(*~
<docu>
	<summary>
			Allows to concat strings using fluent interface. It's similar to C# StringBuilder class
			Usage as follows :
			<code>
				ErrorString := _stringBuilder
					.Clear()
					.Append('Error number: ')
					.Append(INT_TO_STRING(ErrorNumber))
					.Append('. Message: ')
					.Append(ErrorMessage)
					.Append('.')
					.ToString();
			</code>
			
			Inspired by Gerhard Barteling blogpost at https://www.plccoder.com/fluent-code/
	</summary>				
</docu>	
~*)	
FUNCTION_BLOCK StringBuilder
VAR
	{attribute 'hide'}
    _workString:STRING(255);
END_VAR

(*
	Thanks to https://github.com/bengeisler/TcLog
*)

METHOD PROTECTED AnyToString : STRING(255)
VAR_INPUT
	Data:	ANY;
END_VAR
VAR
	pAnyBOOL		: POINTER TO BOOL; 
	pAnyBYTE		: POINTER TO BYTE; 
	pAnyWORD		: POINTER TO WORD; 
	pAnyDWORD		: POINTER TO DWORD;
	pAnyLWORD		: POINTER TO LWORD;
	pAnySINT		: POINTER TO SINT; 
	pAnyUSINT		: POINTER TO USINT;
	pAnyINT			: POINTER TO INT;  
	pAnyUINT		: POINTER TO UINT; 
	pAnyDINT		: POINTER TO DINT; 
	pAnyUDINT		: POINTER TO UDINT;
	pAnyLINT		: POINTER TO LINT; 
	pAnyULINT		: POINTER TO ULINT;
	pAnyLTIME		: POINTER TO LTIME;	
	pAnyReal 		: POINTER TO REAL;
	pAnyLReal		: POINTER TO LREAL;	
	pAnyDateAndTime : POINTER TO DATE_AND_TIME;
	pAnyDate		: POINTER TO DATE;
	pAnyTime		: POINTER TO TIME;
	pAnyWString		: POINTER TO WSTRING;
	pAnyTOD			: POINTER TO TOD;
	pAnyString		: POINTER TO STRING;	
	sString			: T_MAXSTRING;
	wWString		: WSTRING;
END_VAR
IF Data.TypeClass = __SYSTEM.TYPE_CLASS.TYPE_REAL THEN
	pAnyReal := Data.pValue;
	AnyToString := REAL_TO_STRING(pAnyReal^);
	
ELSIF Data.TypeClass = __SYSTEM.TYPE_CLASS.TYPE_LREAL THEN
	pAnyLReal := Data.pValue;
	AnyToString := LREAL_TO_STRING(pAnyLReal^);
	
ELSIF Data.TypeClass = __SYSTEM.TYPE_CLASS.TYPE_DATEANDTIME THEN
	pAnyDateAndTime := Data.pValue;
	AnyToString := DT_TO_STRING(pAnyDateAndTime^);	
	
ELSIF Data.TypeClass = __SYSTEM.TYPE_CLASS.TYPE_DATE THEN
	pAnyDate := Data.pValue;
	AnyToString := DATE_TO_STRING(pAnyDate^);
	
ELSIF Data.TypeClass = __SYSTEM.TYPE_CLASS.TYPE_TIME THEN
	pAnyTime := Data.pValue;
	AnyToString := TIME_TO_STRING(pAnyTime^);
	
ELSIF Data.TypeClass = __SYSTEM.TYPE_CLASS.TYPE_STRING THEN
	pAnyString := Data.pValue;
	AnyToString := pAnyString^;
	
ELSIF Data.TypeClass = __SYSTEM.TYPE_CLASS.TYPE_WSTRING THEN
	pAnyWString := Data.pValue;
	wWString := pAnyWString^;
	WSTRING_TO_STRING2(ADR(sString), ADR(wWstring), SIZEOF(wWString));
	AnyToString := sString;
	
ELSIF Data.TypeClass = __SYSTEM.TYPE_CLASS.TYPE_TIMEOFDAY THEN
	pAnyTOD := Data.pValue;
	AnyToString := TOD_TO_STRING(pAnyTOD^);
ELSIF Data.TypeClass = __SYSTEM.TYPE_CLASS.TYPE_BOOL THEN 	
	pAnyBOOL := Data.pValue;
	AnyToString := BOOL_TO_STRING(pAnyBool^);
ELSIF Data.TypeClass = __SYSTEM.TYPE_CLASS.TYPE_BYTE THEN
	pAnyBYTE := Data.pValue;
	AnyToString := BYTE_TO_STRING(pAnyBYTE^);	
ELSIF Data.TypeClass = __SYSTEM.TYPE_CLASS.TYPE_WORD THEN
	pAnyWORD := Data.pValue;
	AnyToString := WORD_TO_STRING(pAnyWORD^);	
ELSIF Data.TypeClass = __SYSTEM.TYPE_CLASS.TYPE_DWORD THEN
	pAnyDWORD := Data.pValue;	
	AnyToString := DWORD_TO_STRING(pAnyDWORD^);
ELSIF Data.TypeClass = __SYSTEM.TYPE_CLASS.TYPE_LWORD THEN
	pAnyLWORD := Data.pValue;	
	AnyToString := LWORD_TO_STRING(pAnyLWORD^);
ELSIF Data.TypeClass = __SYSTEM.TYPE_CLASS.TYPE_SINT THEN
	pAnySINT := Data.pValue;	
	AnyToString := SINT_TO_STRING(pAnySINT^);					
ELSIF Data.TypeClass = __SYSTEM.TYPE_CLASS.TYPE_USINT THEN
	pAnyUSINT := Data.pValue;	
	AnyToString := USINT_TO_STRING(pAnyUSINT^);	
ELSIF Data.TypeClass = __SYSTEM.TYPE_CLASS.TYPE_INT THEN
	pAnyINT := Data.pValue;	
	AnyToString := INT_TO_STRING(pAnyINT^);	
ELSIF Data.TypeClass = __SYSTEM.TYPE_CLASS.TYPE_UINT THEN
	pAnyUINT := Data.pValue;	
	AnyToString := UINT_TO_STRING(pAnyUINT^);	
ELSIF Data.TypeClass = __SYSTEM.TYPE_CLASS.TYPE_DINT THEN
	pAnyDINT := Data.pValue;	
	AnyToString := DINT_TO_STRING(pAnyDINT^);	
ELSIF Data.TypeClass = __SYSTEM.TYPE_CLASS.TYPE_UDINT THEN
	pAnyUDINT := Data.pValue;	
	AnyToString := UDINT_TO_STRING(pAnyUDINT^);	
ELSIF Data.TypeClass = __SYSTEM.TYPE_CLASS.TYPE_LINT THEN
	pAnyLINT := Data.pValue;	
	AnyToString := LINT_TO_STRING(pAnyLINT^);	
ELSIF Data.TypeClass = __SYSTEM.TYPE_CLASS.TYPE_ULINT THEN
	pAnyULINT := Data.pValue;	
	AnyToString := ULINT_TO_STRING(pAnyULINT^);	
ELSIF Data.TypeClass = __SYSTEM.TYPE_CLASS.TYPE_LTIME THEN
	pAnyLTIME := Data.pValue;	
	AnyToString := LTIME_TO_STRING(pAnyLTIME^);		
ELSE	
	AnyToString := ANY_TO_STRING(Data.pValue^);
END_IF
END_METHOD

METHOD Append : REFERENCE TO StringBuilder
VAR_INPUT
    Text :STRING(255); 
END_VAR
_workString := Concat(_workString,text);
Append REF= THIS^;
END_METHOD

METHOD INTERNAL AppendAny : REFERENCE TO StringBuilder
VAR_INPUT
	Data : ANY;
END_VAR
_workString := Concat(_workString,AnyToString(Data));
AppendAny REF= THIS^;
END_METHOD

METHOD Clear : REFERENCE TO StringBuilder
_workString := '';
Clear REF= THIS^;
END_METHOD

METHOD ToString : STRING(255)
ToString := _workString;
END_METHOD

END_FUNCTION_BLOCK

(* stored: Version 1.1.0.1, ProductVersion 3.1.4024.11
   POU StringBuilder: Id {29d3eafc-7dda-4b19-9304-4e70835541c0}, SpecialFunc None
   Method AnyToString: Id {3d279b77-95bf-47c5-b0be-fcda868e0cb9}
   Method Append: Id {968e12b6-170d-438f-8a91-313208816a32}
   Method AppendAny: Id {48cdce47-2e11-44e0-896c-cc327181b05f}
   Method Clear: Id {3c3bf506-477c-486e-acd4-9a117a320f34}
   Method ToString: Id {e220b688-2381-4979-a1de-20efcbbbfac6} *)
